Universal Robots PolyScope program: DO0.urp

Program DO0 (installation=20240827 directory=/programs createdIn=5.15.1 lastSavedIn=5.15.1 robotSerialNumber=20245500285)
Calibrated DH parameters: a=[0.000097, -0.210459, -0.026602, 0.000137, 0.000078, 0]; d=[0.162601, 254.180657, -54.076236, -199.970743, 0.099615, 0.099684]; alpha=[1.569796, -0.001455, 0.001957, 1.570525, -1.571561, 0]; deltaTheta=[0, -1.053331, 8.839472, -1.50296, 0.000002, 0]
InitVariablesNode
Robot Program (runOnlyOnce=false)
  Script: set_digital_out(0, True )
  Popup Message (haltProgram=false message=True inputType=Text)
  Wait Sleep waitTime=5
  Script: set_digital_out(0, False )
  Popup Message (haltProgram=false message=False inputType=Text)
